PROGRAM MAIN
VAR
	i: INT;
END_VAR

FOR i := 0 TO 20 DO
	GVL_ADS.Array_EPB_TDA_INT[i] := i;
END_FOR

END_PROGRAM

(* stored: Version 1.1.0.1, ProductVersion 3.1.4024.12
   POU MAIN: Id {aa91c11d-963e-430c-9258-5c8b97e79e14}, SpecialFunc None *)
